FUNCTION_BLOCK FB_SaMElementWashing EXTENDS FB_SaMElement
VAR
END_VAR

METHOD FB_init : BOOL
VAR_INPUT
	bInitRetains : BOOL; // if TRUE, the retain variables are initialized (warm start / cold start)
	bInCopyCode : BOOL;  // if TRUE, the instance afterwards gets moved into the copy code (online change)
END_VAR
THIS^.SetText (eLocation := E_BaseLocation.pl, wsDescription := "Mycie");
THIS^.SetText (eLocation := E_BaseLocation.en, wsDescription := "Washing");
THIS^.SetText (eLocation := E_BaseLocation.de, wsDescription := "Waschen");
THIS^.SetName (stName := THIS^.GetTexts ());
END_METHOD

END_FUNCTION_BLOCK

(* stored: Version 1.1.0.1
   POU FB_SaMElementWashing: Id {ef533864-744c-0365-03e8-3819c383dbae}, SpecialFunc None
   Method FB_init: Id {aee59fc8-6814-01af-2dfe-f0bfb60f3f71} *)
